// TwinCAT 3 PLC project Untitled2
// ProgramVersion: 3.1.4024.0
// libraries:
//   Tc2_Standard, * (Beckhoff Automation GmbH)
//   Tc2_System, * (Beckhoff Automation GmbH)
//   Tc3_Module, * (Beckhoff Automation GmbH)
// project tree:
//   / PlcTask.TcTTO
//   POUs/ FB_DataStuff.TcPOU, MAIN.TcPOU
// real-time tasks:
//   TASK PlcTask: cycle T#10ms, priority 20, ADS port 350

CONFIGURATION Untitled2
    RESOURCE PLC ON TwinCAT3
        TASK PlcTask(INTERVAL := T#10ms, PRIORITY := 20);
        PROGRAM MAIN WITH PlcTask : MAIN;
    END_RESOURCE
END_CONFIGURATION

// ---- POUs/MAIN.TcPOU
PROGRAM MAIN

VAR
	fb_HahaDataStuff : FB_DataStuff;
END_VAR

fb_HahaDataStuff();

END_PROGRAM

// ---- POUs/FB_DataStuff.TcPOU
FUNCTION_BLOCK FB_DataStuff

VAR
	a2dArray : ARRAY[1..1000] OF ARRAY[1..3] OF STRING;
	pPointer : POINTER TO ARRAY[1..1000] OF ARRAY[1..3] OF STRING := ADR(a2dArray);
	
	// The value that will be pointed to and calculated amongst the runners
	nValueToCalculate : UINT := 100;
	pPointerToValue : POINTER TO UINT := ADR(nValueToCalculate);
	
	// This will keep track of the index in which the mStoreData method will place data in
	nIndexCounter : UINT := 0;
	
END_VAR

// Pass the pointer to the runner function so it has the direct address of the 2dArray
IF nIndexCounter <> 1000 THEN
		nIndexCounter := nIndexCounter + 1;
	
	mRunnerOne(pDataTable := pPointer^, 
			   nIndexLocation := nIndexCounter,
			   nRunnerValue := pPointerToValue^);
			   
	nIndexCounter := nIndexCounter + 1;
	
	mRunnerOne(pDataTable := pPointer^, 
			   nIndexLocation := nIndexCounter,
			   nRunnerValue := pPointerToValue^);
END_IF

METHOD mRunnerOne : BOOL

VAR_INPUT
	pDataTable : ARRAY[1..1000] OF ARRAY[1..3] OF STRING;
	
	nIndexLocation : UINT;
	nRunnerValue : UINT;
END_VAR

VAR
	nThisRunner : UINT := 1;
	pPointer : POINTER TO ARRAY[1..1000] OF ARRAY[1..3] OF STRING := ADR(pDataTable);
END_VAR
nRunnerValue := nRunnerValue + 1;

mStoreData(pDataTableOp := pPointer^,
		   nIndexToStoreIn := nIndexLocation, 
		   nValue := nRunnerValue, 
		   nRunnerNumber := nThisRunner);
END_METHOD

METHOD mRunnerTwo : BOOL

VAR_INPUT
	pDataTable : ARRAY[1..1000] OF ARRAY[1..3] OF STRING;
	
	nIndexLocation : UINT;
	nRunnerValue : UINT;
END_VAR

VAR
	nThisRunner : UINT := 2;
	pPointer : POINTER TO ARRAY[1..1000] OF ARRAY[1..3] OF STRING := ADR(pDataTable);
END_VAR
nRunnerValue := nRunnerValue - 1;

mStoreData(pDataTableOp := pPointer^,
		   nIndexToStoreIn := nIndexLocation, 
		   nValue := nRunnerValue, 
		   nRunnerNumber := nThisRunner);
END_METHOD

METHOD mStoreData : BOOL

VAR_INPUT
	pDataTableOp : ARRAY[1..1000] OF ARRAY[1..3] OF STRING;
	nIndexToStoreIn : UINT;
	nValue : UINT;
	nRunnerNumber : UINT;
END_VAR

VAR
	sCurrentStringA : STRING;
	sCurrentStringB : STRING;
	pPointerData : POINTER TO ARRAY[1..1000] OF ARRAY[1..3] OF STRING := ADR(pDataTableOp);
END_VAR
// STORES THE CURRENT DATA IN THE ARRAY
sCurrentStringA := UINT_TO_STRING(nValue);
sCurrentStringB := UINT_TO_STRING(nRunnerNumber);

pPointerData^[nIndexToStoreIn][1] := sCurrentStringA;
pPointerData^[nIndexToStoreIn][2] := sCurrentStringB;
END_METHOD

END_FUNCTION_BLOCK
